Staubli VAL3: onF7Event.pgx

program onF7Event()
  local num local1
begin
  // look if the bButton is enable

end
